// TIA Portal project "Hardware" (V14)

(* hardware
DEVICE "ET 200S-Station_1"  ET 200S station
   slot 0: "Baugruppenträger_0"  Rail
   slot 2: "PLC_1"  IM151-8 CPU  6ES7 151-8AB00-0AB0  V2.7
      slot 1: "PROFINET-Schnittstelle_1"  PN-IO
         slot 1: "Port_1"  Port
         slot 2: "Port_2"  Port
         slot 3: "Port_3"  Port
   slot 4: "PM-E 24VDC_1"  PM-E 24VDC  6ES7 138-4CA01-0AA0
   slot 5: "4AI x I 2WIRE ST_1"  4AI x I 2WIRE ST  6ES7 134-4GD00-0AB0
   slot 6: "2AO x U ST_1"  2AO x U ST  6ES7 135-4FB01-0AB0
   slot 7: "8DI x 24VDC_1"  8DI x 24VDC  6ES7 131-4BF00-0AA0
   slot 8: "8DI x 24VDC_2"  8DI x 24VDC  6ES7 131-4BF00-0AA0
   slot 9: "8DI x 24VDC_3"  8DI x 24VDC  6ES7 131-4BF00-0AA0
   slot 10: "8DI x 24VDC_4"  8DI x 24VDC  6ES7 131-4BF00-0AA0
   slot 11: "8DO x 24VDC / 0.5A_1"  8DO x 24VDC / 0.5A  6ES7 132-4BF00-0AA0
   slot 12: "8DO x 24VDC / 0.5A_2"  8DO x 24VDC / 0.5A  6ES7 132-4BF00-0AA0
   slot 13: "8DO x 24VDC / 0.5A_3"  8DO x 24VDC / 0.5A  6ES7 132-4BF00-0AA0
   slot 14: "8DO x 24VDC / 0.5A_4"  8DO x 24VDC / 0.5A  6ES7 132-4BF00-0AA0
DEVICE "HMI_1"  TP 177B 6'' PN/DP
   slot 0: "TP 177B 6'' PN/DP"  TP 177B 6'' PN/DP  6AV6 642-0BA01-1AX1  11.0.2.0
   slot 1: "HMI_RT_1"  TP 177B 6'' PN/DP  6AV6 642-0BA01-1AX1  11.0.2.0
   slot 5: "HMI_1.IE_CP_1"  PROFINET Interface  11.0.0.0
      slot 1: "PROFINET Schnittstelle_1"  PROFINET Interface
         slot 1: "Port_1"  Port
   slot 7: "HMI_1.MPI/DP_CP_1"  MPI/DP Interface  11.0.0.0
DEVICE "S7-1200-Station_1"  S7-1200 Station
   slot 0: "Baugruppenträger_0"  S7-1200 Rack  Rack  V1.0
   slot 1: "PLC_2"  CPU 1214FC DC/DC/DC  6ES7 214-1AF40-0XB0  V4.2
   slot 2: "F-DI 8/16x24VDC_1"  SM 1226 F-DI8/16 x 24VDC  6ES7 226-6BA32-0XB0  V2.0
   slot 3: "AI 1xRTD_1"  AI1 x RTD signal board  6ES7 231-5PA30-0XB0  V2.0
   slot 3: "F-DQ 4x24VDC_1"  SM 1226 F-DQ4 x 24VDC  6ES7 226-6DA32-0XB0  V2.0
   slot 4: "AI 4x13BIT/AQ 2x14BIT_1"  6ES7 234-4HE32-0XB0  V2.0
*)

// ===== PLC "PLC_1"  IM151-8 CPU =====

VAR_GLOBAL   // PLC tag table "Standard-Variablentabelle"
   "n1_sensor" AT %EW128 : Int;
   "n2_sensor" AT %EW132 : Int;
   "n3_press_sensor" AT %EW130 : Int;
END_VAR

ORGANIZATION_BLOCK "Main"   // OB1, FBD
TITLE = "Main Program Sweep (Cycle)"
{ S7_Optimized_Access := 'FALSE' }
VERSION : 0.1
   VAR_TEMP
      OB1_EV_CLASS : Byte;   // Bits 0-3 = 1 (Coming event), Bits 4-7 = 1 (Event class 1)
      OB1_SCAN_1 : Byte;   // 1 (Cold restart scan 1 of OB 1), 3 (Scan 2-n of OB 1)
      OB1_PRIORITY : Byte;   // Priority of OB Execution
      OB1_OB_NUMBR : Byte;   // 1 (Organization block 1, OB1)
      OB1_RESERVED_1 : Byte;   // Reserved for system
      OB1_RESERVED_2 : Byte;   // Reserved for system
      OB1_PREV_CYCLE : Int;   // Cycle time of previous OB1 scan (milliseconds)
      OB1_MIN_CYCLE : Int;   // Minimum cycle time of OB1 (milliseconds)
      test1 : Int;
      OB1_MAX_CYCLE : Int;   // Maximum cycle time of OB1 (milliseconds)
      OB1_DATE_TIME : Date_And_Time;   // Date and time OB1 started
   END_VAR
BEGIN
END_ORGANIZATION_BLOCK

// ===== PLC "PLC_2"  CPU 1214FC DC/DC/DC =====

VAR_GLOBAL   // PLC tag table "Standard-Variablentabelle"
   "high_sensor_s1" AT %EW128 : Int;
   "pressure_sensor_s3" AT %EW130 : Int;
   "high_sensor_s2" AT %EW132 : Int;
END_VAR

DATA_BLOCK "Main_Safety_RTG1_DB"   // DB1, F_DB
{ S7_Optimized_Access := 'TRUE' }
NAME : FUSI
VERSION : 0.1
// stored: InstanceOfName Main_Safety_RTG1
"Main_Safety_RTG1"
BEGIN
END_DATA_BLOCK

DATA_BLOCK "sensor130_to_pa_DB"   // DB2
{ S7_Optimized_Access := 'TRUE' }
VERSION : 0.1
// stored: InstanceOfName sensor130_to_pa
"sensor130_to_pa"
BEGIN
END_DATA_BLOCK

DATA_BLOCK "global_variables"   // DB3
{ S7_Optimized_Access := 'TRUE' }
VERSION : 0.1
   VAR
      density : Real := 1000.0;
      gravity : Real := 9.81;
   END_VAR
BEGIN
END_DATA_BLOCK

DATA_BLOCK "sensor132_to_mm_DB"   // DB4
{ S7_Optimized_Access := 'TRUE' }
VERSION : 0.1
// stored: InstanceOfName sensor132_to_mm
"sensor132_to_mm"
BEGIN
END_DATA_BLOCK

DATA_BLOCK "sensor128_to_mm_DB"   // DB5
{ S7_Optimized_Access := 'TRUE' }
VERSION : 0.1
// stored: InstanceOfName sensor128_to_mm
"sensor128_to_mm"
BEGIN
END_DATA_BLOCK

DATA_BLOCK "Comparing_p3_s1_s2_DB"   // DB6
{ S7_Optimized_Access := 'TRUE' }
VERSION : 0.1
// stored: InstanceOfName Comparing_p3_s1_s2
"Comparing_p3_s1_s2"
BEGIN
END_DATA_BLOCK

FUNCTION_BLOCK "Main_Safety_RTG1"   // FB1, F_FBD
{ S7_Optimized_Access := 'TRUE' }
VERSION : 0.1
BEGIN
END_FUNCTION_BLOCK

FUNCTION_BLOCK "sensor130_to_pa"   // FB2, SCL
{ S7_Optimized_Access := 'TRUE' }
VERSION : 0.1
   VAR_INPUT
      pressure_sensor130 : Real;
   END_VAR
   VAR_OUTPUT
      pressure_pa : Real;
   END_VAR
   VAR_TEMP
      "m" : Real;
      "b" : Real;
   END_VAR
   VAR CONSTANT
      x1 : Real := 0.0;
      x2 : Real := 1011.795;
      y2 : Real := 525.0;
      y1 : Real := -82.0;
   END_VAR
BEGIN

   IF #pressure_sensor130 <= #y1 THEN
       #pressure_pa := 0.0;

   ELSIF #pressure_sensor130 <> 0 AND #pressure_sensor130 > #y1 THEN
       #"m":=(#y2-#y1)/(#x2-#x1);
       #"b" := #y1 - (#"m" * #x1);
       #pressure_pa := ((INT_TO_REAL(#pressure_sensor130)-#"b"))/#"m";
   ELSE
       #pressure_pa := -1.0;
   END_IF;
END_FUNCTION_BLOCK

FUNCTION_BLOCK "sensor132_to_mm"   // FB3, SCL
{ S7_Optimized_Access := 'TRUE' }
VERSION : 0.1
   VAR_INPUT
      high_sensor_s132 : Real;
   END_VAR
   VAR_OUTPUT
      high_sensor_mm : Real;
   END_VAR
   VAR_TEMP
      "m" : Real;
      high_sensor_m : Real;
      "b" : Real;
   END_VAR
   VAR CONSTANT
      x1 : Real := 0.06188348;
      x2 : Real := 0.1031391;
      y1 : Real := 8080.0;
      y2 : Real := 11920.0;
      y0 : Real := -2.0;
   END_VAR
BEGIN

   IF #high_sensor_s132 <= #y0 THEN
       #high_sensor_mm := 0.0;

   ELSIF #high_sensor_s132 <> 0 AND #high_sensor_s132 > #y0 THEN
       #"m":=(#y2-#y1)/(#x2-#x1);
       #"b":=#y1-(#"m"*#x1);
       #high_sensor_m:= ((INT_TO_REAL(#high_sensor_s132)-#"b"))/#"m";
       #high_sensor_mm:=1000*#high_sensor_m;
   ELSE
       #high_sensor_mm := -1.0;
   END_IF;
END_FUNCTION_BLOCK

FUNCTION_BLOCK "sensor128_to_mm"   // FB4, SCL
{ S7_Optimized_Access := 'TRUE' }
VERSION : 0.1
   VAR_INPUT
      high_sensor_s128 : Real;
   END_VAR
   VAR_OUTPUT
      high_sensor_mm : Real;
   END_VAR
   VAR_TEMP
      "m" : Real;
      high_sensor_m : Real;
      "b" : Real;
   END_VAR
   VAR CONSTANT
      x1 : Real := 0.0;
      x2 : Real := 0.1031391;
      y2 : Real := 973.0;
      y1 : Real := 560.0;
   END_VAR
BEGIN

   IF #high_sensor_s128 <= #y1 THEN
       #high_sensor_mm := 0.0;

   ELSIF #high_sensor_s128 <> 0 AND #high_sensor_s128 > #y1 THEN
       #"m":=(#y2-#y1)/(#x2-#x1);
       #"b" := #y1 - (#"m" * #x1);
       #high_sensor_m:= ((INT_TO_REAL(#high_sensor_s128)-#"b"))/#"m";
       #high_sensor_mm:=1000*#high_sensor_m;
   ELSE
       #high_sensor_mm := -1.0;
   END_IF;
END_FUNCTION_BLOCK

FUNCTION_BLOCK "Comparing_p3_s1_s2"   // FB5, SCL
{ S7_Optimized_Access := 'TRUE' }
VERSION : 0.1
   VAR_INPUT
      h_from_pressure130 : Real;
      h_from_high128 : Real;
      h_from_high132 : Real;
   END_VAR
   VAR_OUTPUT
      difference1_mm_130_132 : Real;
      difference1_percentage_130_132 : Real;
      difference2_mm_132_128 : Real;
      difference2_percentage_132_128 : Real;
   END_VAR
BEGIN
   IF #h_from_pressure130 <> 0 THEN
       #difference1_mm_130_132 := #h_from_pressure130 - #h_from_high132;
       #difference1_percentage_130_132 := 100 * (#h_from_pressure130 - #h_from_high132) / #h_from_pressure130;
   END_IF;

   IF #h_from_high132 <> 0 THEN
       #difference2_mm_132_128 := #h_from_high132 - #h_from_high128;
       #difference2_percentage_132_128 := 100 * (#h_from_high132 - #h_from_high128) / #h_from_high132;
   END_IF;
END_FUNCTION_BLOCK

FUNCTION "test_Vergleichen" : Void   // FC1, FBD
{ S7_Optimized_Access := 'FALSE' }
VERSION : 0.1
   VAR_INPUT
      n1_sensor : Int;
   END_VAR
   VAR_OUTPUT
      n1_wert : Int;
   END_VAR
BEGIN

REGION Network 1
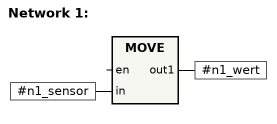
   #n1_wert := #n1_sensor;
END_REGION
END_FUNCTION

FUNCTION "pressure_to_h_mm" : Void   // FC2, SCL
{ S7_Optimized_Access := 'TRUE' }
VERSION : 0.1
   VAR_INPUT
      pressure : Real;
   END_VAR
   VAR_OUTPUT
      h_by_sensorpress_mm : Real;
   END_VAR
BEGIN
   #h_by_sensorpress_mm := #pressure*1000 / ("global_variables".density * "global_variables".gravity);
END_FUNCTION

ORGANIZATION_BLOCK "Main"   // OB1, FBD, ProgramCycle
TITLE = "Main Program Sweep (Cycle)"
{ S7_Optimized_Access := 'TRUE' }
VERSION : 0.1
   VAR_INPUT
      Initial_Call : Bool;   // Initial call of this OB
      Remanence : Bool;   // =True, if remanent data are available
   END_VAR
   VAR_TEMP
      s3_pressure_pa : Real;
      s3_high_container_mm : Real;
      s1_high128_mm : Real;
      s2_high132_mm : Real;
      diff1_p_130_132 : Real;
      diff1_mm_130_132 : Real;
      diff2_mm_128_132 : Real;
      diff2_p_128_132 : Real;
      test1 : Int;
      test2 : Int;
      test3 : Int;
   END_VAR
BEGIN

REGION Network 1
   // high sensor 1 128
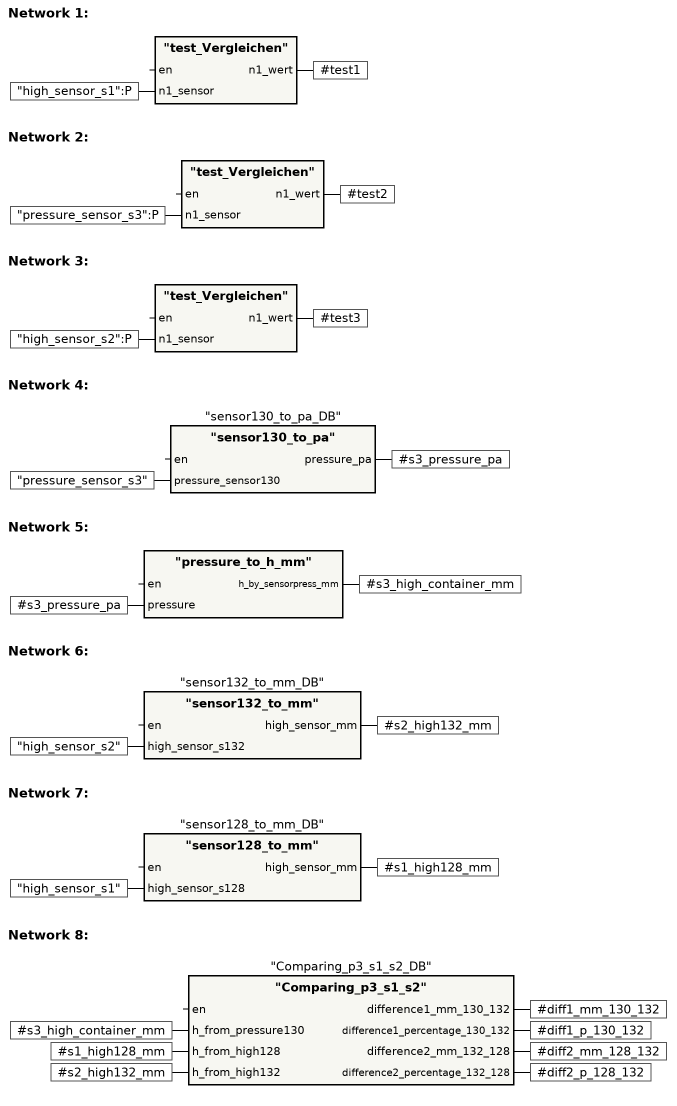
   "test_Vergleichen"(n1_sensor := "high_sensor_s1":P, n1_wert => #test1);
END_REGION

REGION Network 2
   // high sensor pressure
   "test_Vergleichen"(n1_sensor := "pressure_sensor_s3":P, n1_wert => #test2);
END_REGION

REGION Network 3
   // high sensor 2 132
   "test_Vergleichen"(n1_sensor := "high_sensor_s2":P, n1_wert => #test3);
END_REGION

REGION Network 4
   "sensor130_to_pa_DB"(pressure_sensor130 := "pressure_sensor_s3", pressure_pa => #s3_pressure_pa);   // "sensor130_to_pa"
END_REGION

REGION Network 5
   "pressure_to_h_mm"(pressure := #s3_pressure_pa, h_by_sensorpress_mm => #s3_high_container_mm);
END_REGION

REGION Network 6
   "sensor132_to_mm_DB"(high_sensor_s132 := "high_sensor_s2", high_sensor_mm => #s2_high132_mm);   // "sensor132_to_mm"
END_REGION

REGION Network 7
   "sensor128_to_mm_DB"(high_sensor_s128 := "high_sensor_s1", high_sensor_mm => #s1_high128_mm);   // "sensor128_to_mm"
END_REGION

REGION Network 8
   "Comparing_p3_s1_s2_DB"(h_from_pressure130 := #s3_high_container_mm,   // "Comparing_p3_s1_s2"
                           h_from_high128 := #s1_high128_mm,
                           h_from_high132 := #s2_high132_mm,
                           difference1_mm_130_132 => #diff1_mm_130_132,
                           difference1_percentage_130_132 => #diff1_p_130_132,
                           difference2_mm_132_128 => #diff2_mm_128_132,
                           difference2_percentage_132_128 => #diff2_p_128_132);
END_REGION
END_ORGANIZATION_BLOCK

(* ===== HMI "HMI_RT_1" =====
system functions are stored by id; their names below are inferred from use
connection "HMI_Verbindung_1": ETHERNET, SIMATIC S7 300/400 MPI
connection "HMI_Verbindung_2": ETHERNET, SIMATIC S7 1200

HMI tags "Standard-Variablentabelle"
   "Variable_Bildnummer" : UInt, internal
   "A_rot" : Bool = PLC A_rot AT %A9.6, 1 s
   "A_gelb" : Bool = PLC A_gelb AT %A9.7, 1 s
   "A_gruen" : Bool = PLC A_gruen AT %A10.0, 1 s
   "F_gruen" : Bool = PLC F_gruen AT %A10.7, 1 s
   "F_rot" : Bool = PLC F_rot AT %A10.6, 1 s
   "Variable_Tag_H" : Int = PLC Variable.Tag_H AT %DB200.DBW16, 1 s
   "Variable_Tag_M" : Int = PLC Variable.Tag_M AT %DB200.DBW18, 1 s
   "Variable_Nacht_H" : Int = PLC Variable.Nacht_H AT %DB200.DBW22, 1 s
   "Variable_Nacht_M" : Int = PLC Variable.Nacht_M AT %DB200.DBW24, 1 s
   "Variable_Abstand" : Real = PLC Variable.Abstand AT %DB200.DBD0, 1 s
   "Farben_Rot" : Real = PLC Farben.Rot AT %DB4.DBD120, 1 s
   "Farben_Blau" : Real = PLC Farben.Blau AT %DB4.DBD124, 1 s
   "Farben_Gelb" : Real = PLC Farben.Gelb AT %DB4.DBD128, 1 s
   "Farben_index" : Int = PLC Farben.index AT %DB4.DBW132, 1 s
   "Farben_schreiben" : Bool = PLC Farben.schreiben AT %DB4.DBX134.0, 1 s
   "DB3_Farben_rot" : Int = PLC DB3_Farben.rot AT %DB3.DBW0, 1 s
   "DB3_Farben_blau" : Int = PLC DB3_Farben.blau AT %DB3.DBW4, 1 s
   "Von_300_Gewicht_rot" : Real = PLC Von_300.Gewicht_rot AT %DB100.DBD0, 1 s
   "Von_300_Gewicht_Gruen" : Real = PLC Von_300.Gewicht_Gruen AT %DB100.DBD4, 1 s
   "Von_300_Gewicht_blau" : Real = PLC Von_300.Gewicht_blau AT %DB100.DBD8, 1 s
   "Zu_1200_Gewicht_Gruen" : Real = PLC Zu_1200.Gewicht_Gruen AT %DB100.DBD4, 1 s
   "Zu_1200_Gewicht_rot" : Real = PLC Zu_1200.Gewicht_rot AT %DB100.DBD0, 1 s
   "Zu_1200_Gewicht_Blau" : Real = PLC Zu_1200.Gewicht_Blau AT %DB100.DBD8, 1 s
   "DB3_Farben_gruen" : Int = PLC DB3_Farben.gruen AT %DB3.DBW2, 1 s

text list "Textliste_Bildnamen": 1 'Grundbild / base image'; 2 'Ampel / Trafic light'; 3 'Uhrzeit / Time'

text list "Farben": 0 'Orange'; 1 'Violett'; 2 'Hellblau'

screen "Grundbild" 320x200, template "Vorlage_1"
   on GenerateScreen: SetTag("Variable_Bildnummer", 1)
   TextField "HmiScreenItemData" at 21,55 size 179x36; Text 'Willkommen zum HMI_1 (TP 177B 6″ PN/DP)!'
   Button "Ampel" at 1,1 size 104x36; TextOff 'Ampel / Trafic light'
      on Release: ActivateScreen("Ampel", 0)
   Button "Uhrzeit" at 106,1 size 104x36; TextOff 'Uhrzeit / Time'
      on Release: ActivateScreen("Uhrzeit", 0)
   TextField "Textfeld_1" at 243,9 size 51x20; Text 'Sprache'
   Button "Schaltfläche_1" at 228,30 size 80x25; TextOff 'Deutsch'
      on Release: function_fb9197e8(L de-DE)
   Button "Schaltfläche_2" at 228,56 size 80x25; TextOff 'English'
      on Release: function_fb9197e8(L en-US)
   Button "Schaltfläche_3" at 0,124 size 160x25; TextOff 'Farben'
      on Click: ActivateScreen("Farben", 0)

Template "Vorlage_1" 320x200
   Button "Beenden" at 267,150 size 51x47; TextOff 'Beenden / Operate'; TextOn 'Beenden / Finish'; PictureOff "ExitRuntime_TP_177B_6_PNDP"; PictureOn "ExitRuntime_TP_177B_6_PNDP"
      on Release: StopRuntime(0)
   Button "Template_Button" at 214,150 size 51x47; TextOff 'Text'
   Button "Template_Button_1" at 160,150 size 51x47; TextOff 'Text'
   Button "Template_Button_2" at 107,150 size 51x47; TextOff 'Text'
   Button "Template_Button_3" at 54,150 size 51x47; TextOff 'Text'
   Button "Startbild" at 1,150 size 51x47; TextOff 'Startbild / Home'; PictureOff "NavigateHome_TP_177B_6_PNDP"; PictureOn "NavigateHome_TP_177B_6_PNDP"
      on Release: ActivateScreen("Grundbild", 0)

screen "Ampel" 320x200, template "Vorlage_1"
   on GenerateScreen: SetTag("Variable_Bildnummer", 2)
   GraphicView "Grafikanzeige_1" at 0,1 size 319x148; Picture "strasse"
   Group "Group" at 170,4 size 60x25
   Group "Group_1" at 83,119 size 60x25
   Group "Group_2" at 188,106 size 25x43
   Group "Group_3" at 110,1 size 25x43
   Circle "Kreis_1" at 173,7 size 18x18
      Visibility <- "A_rot"
   Circle "Kreis_2" at 192,7 size 18x18
      Appearance <- "A_gelb"
   Circle "Kreis_3" at 211,8 size 18x18
      Visibility <- "A_gruen"
   Circle "Kreis_4" at 122,122 size 18x18
      Visibility <- "A_rot"
   Circle "Kreis_5" at 103,122 size 18x18
      Appearance <- "A_gelb"
   Circle "Kreis_6" at 84,123 size 18x18
      Visibility <- "A_gruen"
   Circle "Kreis_9" at 192,107 size 18x18
      Visibility <- "F_gruen"
   Circle "Kreis_7" at 192,127 size 18x18
      Visibility <- "F_rot"
   Circle "Kreis_8" at 114,25 size 18x18
      Visibility <- "F_gruen"
   Circle "Kreis_10" at 114,5 size 18x18
      Visibility <- "F_rot"

screen "Uhrzeit" 320x200, template "Vorlage_1"
   on GenerateScreen: SetTag("Variable_Bildnummer", 3)
   Button "Zurück" at 1,1 size 104x36; TextOff 'Zurück / back'
      on Release: ActivateScreen("Grundbild", 0)
   TextField "Textfeld_1" at 18,42 size 31x20; Text 'Tag: / day'
   IOField "EA-Feld_1" at 60,42 size 17x20; FormatPattern 99
      ProcessValue <- "Variable_Tag_H"
   TextField "Textfeld_2" at 77,42 size 10x20; Text ':'
   IOField "EA-Feld_2" at 87,42 size 17x20; FormatPattern 99
      ProcessValue <- "Variable_Tag_M"
   TextField "Textfeld_3" at 105,42 size 42x20; Text 'Uhr / o'clock'
   TextField "Textfeld_4" at 19,72 size 41x20; Text 'Nacht: / night'
   IOField "EA-Feld_3" at 61,72 size 17x20; FormatPattern 99
      ProcessValue <- "Variable_Nacht_H"
   TextField "Textfeld_5" at 78,72 size 10x20; Text ':'
   IOField "EA-Feld_4" at 88,72 size 17x20; FormatPattern 99
      ProcessValue <- "Variable_Nacht_M"
   TextField "Textfeld_6" at 106,72 size 42x20; Text 'Uhr / o'clock'

screen "Abstandbild" 320x200
   Gauge "Zeigerinstrument_1" at 114,0 size 200x200; CaptionText 'Abstand'; UnitText 'mm'
      ProcessValue <- "Variable_Abstand"
   Button "Schaltfläche_1" at 5,167 size 80x25; TextOff 'Grundbild'

screen "Farben" 320x200
   Button "Schaltfläche_1" at 0,176 size 150x24; TextOff 'Grundbild'
      on Click: ActivateScreen("Grundbild", 0)
   TextField "Textfeld_1" at 19,20 size 29x20; Text 'Rot'
   TextField "Textfeld_2" at 19,44 size 29x20; Text 'Blau'
   TextField "Textfeld_3" at 19,73 size 29x20; Text 'Gelb'
   TextField "Textfeld_4" at 19,99 size 35x20; Text 'Index'
   IOField "EA-Feld_1" at 54,20 size 80x20; FormatPattern s999999999.999
      ProcessValue <- "Farben_Rot"
   IOField "EA-Feld_2" at 54,48 size 80x20; FormatPattern s999999999.999
      ProcessValue <- "Farben_Blau"
   IOField "EA-Feld_3" at 54,75 size 80x20; FormatPattern s999999999.999
      ProcessValue <- "Farben_Gelb"
   IOField "EA-Feld_4" at 54,100 size 80x20; FormatPattern s99999
      ProcessValue <- "Farben_index"
   Button "Schaltfläche_2" at 56,134 size 80x25; TextOff 'Schreiben'
      on Click: InvertBit("Farben_schreiben")
      Appearance <- "Farben_schreiben"
   SymbolicIOField "Symbolisches EA-Feld_1" at 145,100 size 119x22; TextOff '0'; TextOn '1'; TextList "Farben"
      ProcessValue <- "Farben_index"

screen "Kontrollbild" 320x200
   TextField "Textfeld_1" at 13,28 size 30x20; Text 'grun'
   TextField "Textfeld_2" at 144,28 size 82x20; Text 'ausgabe grun'
   TextField "Textfeld_3" at 14,53 size 29x20; Text 'rot'
   TextField "Textfeld_4" at 13,79 size 29x20; Text 'Blau'
   TextField "Textfeld_5" at 147,80 size 81x20; Text 'Ausgabe Blau'
   TextField "Textfeld_6" at 146,52 size 75x20; Text 'ausgabe Rot'
   IOField "EA-Feld_2" at 228,52 size 80x20; FormatPattern s999999999.999
      ProcessValue <- "Von_300_Gewicht_rot"
   IOField "EA-Feld_3" at 229,27 size 80x20; FormatPattern s999999999.999
      ProcessValue <- "Von_300_Gewicht_Gruen"
   IOField "EA-Feld_4" at 229,81 size 80x20; FormatPattern s999999999.999
      ProcessValue <- "Von_300_Gewicht_blau"
   IOField "EA-Feld_1" at 47,30 size 93x20; FormatPattern s99999
      ProcessValue <- "DB3_Farben_gruen"
   IOField "EA-Feld_5" at 46,53 size 94x20; FormatPattern s99999
      ProcessValue <- "DB3_Farben_rot"
   IOField "EA-Feld_6" at 46,80 size 95x20; FormatPattern s99999
      ProcessValue <- "DB3_Farben_blau"
*)